PROGRAM MAIN
VAR_INPUT
	Axis_S				: FBCylTronicCylinder;
	Axis_T				: FBCyltronicCylinder;
	Axis_R				: FBCyltronicCylinder;
	rSetPos_R			: REAL := 0;
	rSetPos_S			: REAL := 0;
	rSetPos_T			: REAL := 0;
END_VAR

VAR
	Sinus				: FB_CTRL_SIGNAL_GENERATOR;
	SinusParams			: ST_CTRL_SIGNAL_GENERATOR_PARAMS;
	SinusMode			: E_CTRL_MODE := E_CTRL_MODE.eCTRL_MODE_ACTIVE;
	rXBallPos			: REAL; //Ball Position X Axis in mm
	rYBallPos			: REAL; //Ball Position Y Axis in mm
	rMaxTouchPos		: REAL := 363 / 2;
	rSetVelo			: REAL := 300;
	rSetAcc				: REAL := 5;
	rSetForce			: REAL := 800;
	Modus				: Mode;
	trigDown, trigUp	: R_TRIG;
	bDOWN, bUp			: BOOL;
	bBallOnPlate		: BOOL;
	bBallonPlateButton	: BOOL := FALSE;
	FB_FigureGenerator	: FB_FigureGenerator;
END_VAR

Axis_R(stAxisName:='Achse 1');
Axis_S(stAxisName:='Achse 2');
Axis_T(stAxisName:='Achse 3');
Touchpanel();
AC_ModeSelection();
AC_TouchPos();
CONTROLLER();
FB_FigureGenerator();

ACTION AC_ModeSelection:

//Ausschaltbedingungen (Prio 1)
IF NOT gvl.Einbefehl OR NOT gvl.NOTAUS THEN
	Axis_R.bEnable := FALSE;
	Axis_S.bEnable := FALSE;
	Axis_T.bEnable := FALSE;
	Modus := Mode.Off;
	GVL.V48Einbefehl := FALSE;
END_IF

IF NOT GVL.NOTAUS THEN
	GVL.Einbefehl := FALSE;
END_IF

//Resetbefehl
IF gvl.reset THEN
	Axis_R.bReset := TRUE;
	Axis_S.bReset := TRUE;
	Axis_T.bReset := TRUE;
	Modus := Mode.Off;
END_IF

Axis_R.rSetForce	:= rSetForce;
Axis_S.rSetForce	:= rSetForce;
Axis_T.rSetForce	:= rSetForce;
Axis_R.rSetAcc		:= rSetAcc;
Axis_S.rSetAcc		:= rSetAcc;
Axis_T.rSetAcc		:= rSetAcc;
Axis_R.rSetVelo		:= rSetVelo;
Axis_S.rSetVelo		:= rSetVelo;
Axis_T.rSetVelo		:= rSetVelo;
Axis_R.bHoming 		:= FALSE;
Axis_S.bHoming 		:= FALSE;
Axis_T.bHoming 		:= FALSE;

IF (NOT Axis_R.Ready OR NOT Axis_S.Ready OR NOT Axis_T.Ready) AND gvl.Einbefehl AND gvl.NOTAUS THEN
	GVL.V48Einbefehl := TRUE;
	Modus := Mode.Homing;
ELSIF GVL.Grundposition THEN
	Modus := Mode.Position;
ELSIF gvl.BndP THEN
	Modus:=Mode.BallundPlate;
ELSIF gvl.Sinus THEN
	Modus:=Mode.Sinus;
ELSIF GVL.Tilt THEN
	Modus:=Mode.Tilt;
ELSIF gvl.Homing THEN
	Modus:=Mode.Homing;
END_IF

GVL.Sinus_Aktiv := FALSE;
GVL.BNP_Aktiv	:= FALSE;
IF Modus <> Mode.BallundPlate THEN
	bBallOnPlateButton := FALSE;
	bBallOnPlate := FALSE;
END_IF

CASE Modus OF
	Mode.Off:
		;
		
	Mode.Homing:
		Axis_R.bEnable := TRUE;
		Axis_S.bEnable := TRUE;
		Axis_T.bEnable := TRUE;
		Axis_R.bHoming := TRUE;
		Axis_S.bHoming := TRUE;
		Axis_T.bHoming := TRUE;
		gvl.eingabesperre:=TRUE;
		
	Mode.Position:
		IF gvl.Automatik THEN
			rSetPos_R := rSetPos_S := rSetPos_T	:= gvl.Eingabe_Sollposition;
		END_IF
	
	Mode.Tilt:
		;
	
	Mode.Sinus:
		SinusParams.eSignalType := E_CTRL_SIGNAL_TYPE.eCTRL_SINUS;
		SinusParams.fAmplitude := (MaxTravel - 2 ) / 2;
		SinusParams.fOffset := MaxTravel / 2;
		SinusParams.tCtrlCycleTime := T#2MS;
		SinusParams.tCylceDuration := T#2S;
		SinusParams.tTaskCycleTime := T#2MS;
		Sinus(stParams := SinusParams);
		Sinus.eMode := SinusMode;
		rSetPos_R := rSetPos_S := rSetPos_T := LREAL_TO_REAL(Sinus.fOut);
	
	Mode.BallundPlate:
		bBallOnPlate := bBallOnPlateButton;
	
		;
END_CASE
Axis_R.rSetPos	:= rSetPos_R;
Axis_S.rSetPos	:= rSetPos_S;
Axis_T.rSetPos	:= rSetPos_T;
END_ACTION

ACTION AC_TouchPos:
IF CONTROLLER.bReAktiv THEN
	rXBallPos := Touchpanel.touch_scale_x.rX_mm;
	rYBallPos := Touchpanel.touch_scale_y.rX_mm;
ELSE
	rXBallPos := -180;
	rYBallPos := -142;
END_IF
END_ACTION

END_PROGRAM

(* stored: Version 1.1.0.1, ProductVersion 3.1.4024.12
   POU MAIN: Id {60bc0b30-1cdb-42b0-8bc7-ac64af597b82}, SpecialFunc None
   Action AC_ModeSelection: Id {2f31f6c9-d783-4214-bd42-62c52be136ef}
   Action AC_TouchPos: Id {a5abb554-29a7-45b2-a1a8-90708d4f4208} *)
